// TwinCAT 3 PLC project Nepionic_PackML
// Title: Nepionic_PackML
// Company: Nepionic
// Author: Nepionic
// ProjectVersion: 0.1.1
// ProgramVersion: 3.1.4026.21
// libraries:
//   Nepionic_Log, * (Nepionic)
//   Tc2_System, * (Beckhoff Automation GmbH)
// project tree:
//   Commands/Generic/ ActionStateCommands.TcIO, HoldableStateCommands.TcIO, ClearedStateCommands.TcIO, ResettableStateCommands.TcIO, RunningStateCommands.TcIO
//   Commands/ AbortedCommands.TcIO, AbortingCommands.TcIO, ClearingCommands.TcIO, CompletedCommands.TcIO, CompletingCommands.TcIO, ExecuteCommands.TcIO, HeldCommands.TcIO, HoldingCommands.TcIO, IdleCommands.TcIO, ResettingCommands.TcIO, StartingCommands.TcIO, StoppedCommands.TcIO, StoppingCommands.TcIO, SuspendedCommands.TcIO, SuspendingCommands.TcIO, UnholdingCommands.TcIO, UnsuspendingCommands.TcIO
//   StateMachine/ State.TcDUT, StateMachine.TcPOU
//   UnitMode/ UnitMode.TcIO, DefaultUnitMode.TcPOU

// ---- StateMachine/State.TcDUT
{attribute 'qualified_only'}
{attribute 'strict'}
{attribute 'to_string'}
TYPE State :
(
	Undefined := 0,
    Clearing := 1,
    Stopped := 2,
    Starting := 3,
    Idle := 4,
    Suspended := 5,
	Execute := 6,
    Stopping := 7,
    Aborting := 8,
    Aborted := 9,
    Holding := 10,
    Held := 11,
    Unholding := 12,
    Suspending := 13,
    Unsuspending := 14,
    Resetting := 15,
    Completing := 16,
    Completed := 17
);
END_TYPE

// ---- Commands/Generic/ActionStateCommands.TcIO
INTERFACE PUBLIC ActionStateCommands EXTENDS __System.IQueryInterface

METHOD PUBLIC StateComplete
END_METHOD

END_INTERFACE

// ---- Commands/Generic/HoldableStateCommands.TcIO
INTERFACE PUBLIC HoldableStateCommands EXTENDS __System.IQueryInterface

METHOD PUBLIC Hold
END_METHOD

END_INTERFACE

// ---- Commands/Generic/ClearedStateCommands.TcIO
INTERFACE PUBLIC ClearedStateCommands EXTENDS __System.IQueryInterface

METHOD PUBLIC Abort
END_METHOD

END_INTERFACE

// ---- Commands/Generic/ResettableStateCommands.TcIO
INTERFACE PUBLIC ResettableStateCommands EXTENDS __System.IQueryInterface

METHOD PUBLIC Reset
END_METHOD

END_INTERFACE

// ---- Commands/Generic/RunningStateCommands.TcIO
INTERFACE PUBLIC RunningStateCommands EXTENDS ClearedStateCommands

METHOD PUBLIC Stop
END_METHOD

END_INTERFACE

// ---- Commands/AbortedCommands.TcIO
INTERFACE PUBLIC AbortedCommands EXTENDS __System.IQueryInterface

METHOD PUBLIC Clear
END_METHOD

END_INTERFACE

// ---- Commands/AbortingCommands.TcIO
INTERFACE PUBLIC AbortingCommands EXTENDS ActionStateCommands

END_INTERFACE

// ---- Commands/ClearingCommands.TcIO
INTERFACE PUBLIC ClearingCommands EXTENDS ClearedStateCommands, ActionStateCommands

END_INTERFACE

// ---- Commands/CompletedCommands.TcIO
INTERFACE PUBLIC CompletedCommands EXTENDS RunningStateCommands, ResettableStateCommands

END_INTERFACE

// ---- Commands/CompletingCommands.TcIO
INTERFACE PUBLIC CompletingCommands EXTENDS RunningStateCommands, ActionStateCommands

END_INTERFACE

// ---- Commands/ExecuteCommands.TcIO
INTERFACE PUBLIC ExecuteCommands EXTENDS RunningStateCommands, ActionStateCommands, HoldableStateCommands

METHOD PUBLIC Suspend
END_METHOD

END_INTERFACE

// ---- Commands/HeldCommands.TcIO
INTERFACE PUBLIC HeldCommands EXTENDS RunningStateCommands

METHOD PUBLIC Unhold
END_METHOD

END_INTERFACE

// ---- Commands/HoldingCommands.TcIO
INTERFACE PUBLIC HoldingCommands EXTENDS RunningStateCommands, ActionStateCommands

END_INTERFACE

// ---- Commands/IdleCommands.TcIO
INTERFACE PUBLIC IdleCommands EXTENDS RunningStateCommands

METHOD PUBLIC Start
END_METHOD

END_INTERFACE

// ---- Commands/ResettingCommands.TcIO
INTERFACE PUBLIC ResettingCommands EXTENDS RunningStateCommands, ActionStateCommands

END_INTERFACE

// ---- Commands/StartingCommands.TcIO
INTERFACE PUBLIC StartingCommands EXTENDS RunningStateCommands, ActionStateCommands, HoldableStateCommands

END_INTERFACE

// ---- Commands/StoppedCommands.TcIO
INTERFACE PUBLIC StoppedCommands EXTENDS ClearedStateCommands, ResettableStateCommands

END_INTERFACE

// ---- Commands/StoppingCommands.TcIO
INTERFACE PUBLIC StoppingCommands EXTENDS ClearedStateCommands, ActionStateCommands

END_INTERFACE

// ---- Commands/SuspendedCommands.TcIO
INTERFACE PUBLIC SuspendedCommands EXTENDS RunningStateCommands, HoldableStateCommands

METHOD PUBLIC Unsuspend
END_METHOD

END_INTERFACE

// ---- Commands/SuspendingCommands.TcIO
INTERFACE PUBLIC SuspendingCommands EXTENDS RunningStateCommands, ActionStateCommands, HoldableStateCommands

END_INTERFACE

// ---- Commands/UnholdingCommands.TcIO
INTERFACE PUBLIC UnholdingCommands EXTENDS RunningStateCommands, ActionStateCommands, HoldableStateCommands

END_INTERFACE

// ---- Commands/UnsuspendingCommands.TcIO
INTERFACE PUBLIC UnsuspendingCommands EXTENDS RunningStateCommands, ActionStateCommands, HoldableStateCommands

END_INTERFACE

// ---- UnitMode/UnitMode.TcIO
INTERFACE PUBLIC UnitMode

METHOD PUBLIC Abort
END_METHOD

METHOD PUBLIC Clear
END_METHOD

{attribute 'monitoring':='call'}
PROPERTY PUBLIC CurrentState : State
GET
END_GET
END_PROPERTY

METHOD PUBLIC CyclicCall
END_METHOD

METHOD PUBLIC Hold
END_METHOD

{attribute 'monitoring':='call'}
PROPERTY PUBLIC IsAborted : BOOL
GET
END_GET
END_PROPERTY

{attribute 'monitoring':='call'}
PROPERTY PUBLIC IsAborting : BOOL
GET
END_GET
END_PROPERTY

{attribute 'monitoring':='call'}
PROPERTY PUBLIC IsClearing : BOOL
GET
END_GET
END_PROPERTY

{attribute 'monitoring':='call'}
PROPERTY PUBLIC IsCompleted : BOOL
GET
END_GET
END_PROPERTY

{attribute 'monitoring':='call'}
PROPERTY PUBLIC IsCompleting : BOOL
GET
END_GET
END_PROPERTY

{attribute 'monitoring':='call'}
PROPERTY PUBLIC IsExecuting : BOOL
GET
END_GET
END_PROPERTY

{attribute 'monitoring':='call'}
PROPERTY PUBLIC IsHeld : BOOL
GET
END_GET
END_PROPERTY

{attribute 'monitoring':='call'}
PROPERTY PUBLIC IsHolding : BOOL
GET
END_GET
END_PROPERTY

{attribute 'monitoring':='call'}
PROPERTY PUBLIC IsIdle : BOOL
GET
END_GET
END_PROPERTY

{attribute 'monitoring':='call'}
PROPERTY PUBLIC IsResetting : BOOL
GET
END_GET
END_PROPERTY

{attribute 'monitoring':='call'}
PROPERTY PUBLIC IsStarting : BOOL
GET
END_GET
END_PROPERTY

{attribute 'monitoring':='call'}
PROPERTY PUBLIC IsStopped : BOOL
GET
END_GET
END_PROPERTY

{attribute 'monitoring':='call'}
PROPERTY PUBLIC IsStopping : BOOL
GET
END_GET
END_PROPERTY

{attribute 'monitoring':='call'}
PROPERTY PUBLIC IsSuspended : BOOL
GET
END_GET
END_PROPERTY

{attribute 'monitoring':='call'}
PROPERTY PUBLIC IsSuspending : BOOL
GET
END_GET
END_PROPERTY

{attribute 'monitoring':='call'}
PROPERTY PUBLIC IsUnholding : BOOL
GET
END_GET
END_PROPERTY

{attribute 'monitoring':='call'}
PROPERTY PUBLIC IsUnsuspending : BOOL
GET
END_GET
END_PROPERTY

METHOD PUBLIC Reset
END_METHOD

METHOD PUBLIC Start
END_METHOD

METHOD PUBLIC Stop
END_METHOD

METHOD PUBLIC Suspend
END_METHOD

METHOD PUBLIC Unhold
END_METHOD

METHOD PUBLIC Unsuspend
END_METHOD

END_INTERFACE

// ---- StateMachine/StateMachine.TcPOU
{attribute 'linkalways'} 
{attribute 'no_explicit_call' := 'This FB is a CLASS and must be accessed using methods or properties'}
{attribute 'enable_dynamic_creation'}
FUNCTION_BLOCK PUBLIC StateMachine
VAR_GENERIC CONSTANT
	initial_state : State := State.Idle;
END_VAR
IMPLEMENTS
	AbortingCommands,
	ClearingCommands,
	HeldCommands,
	CompletingCommands,
	ExecuteCommands,
	AbortedCommands,
	CompletedCommands,
	HoldingCommands,
	UnsuspendingCommands,
	UnholdingCommands,
	SuspendingCommands,
	SuspendedCommands,
	IdleCommands,
	ResettingCommands,
	StartingCommands,
	StoppedCommands,
	StoppingCommands
VAR
	current_state : State := initial_state;
	logger : DefaultLogger(__POUNAME());
END_VAR

METHOD PUBLIC Abort
IF IsAborting OR IsAborted THEN
	RETURN;
END_IF

logger.Debug('Abort() called, aborting');
ChangeState(State.Aborting);
END_METHOD

METHOD PRIVATE ChangeState
VAR_INPUT
	state : State;
END_VAR
logger
	.WithIntAttribute('exiting_state', current_state)
	.WithIntAttribute('entering_state', state)
	.Debug('Changing state');

current_state := state;
END_METHOD

METHOD PUBLIC Clear
IF IsAborted THEN
	logger.Debug('Clear() called, clearing');
	ChangeState(State.Clearing);
END_IF
END_METHOD

{attribute 'monitoring':='call'}
PROPERTY PUBLIC CurrentState : State
GET
CurrentState := current_state;
END_GET
END_PROPERTY

METHOD PUBLIC Hold
CASE current_state OF
	State.Execute,
	State.Starting,
	State.Suspending,
	State.Suspended,
	State.Unsuspending,
	State.Unholding:
		logger.Debug('Hold() called, holding');
		ChangeState(State.Holding);	
END_CASE
END_METHOD

{attribute 'monitoring':='call'}
PROPERTY PUBLIC IsAborted : BOOL
GET
IsAborted := (current_state = State.Aborted);
END_GET
END_PROPERTY

{attribute 'monitoring':='call'}
PROPERTY PUBLIC IsAborting : BOOL
GET
IsAborting := (current_state = State.Aborting);
END_GET
END_PROPERTY

{attribute 'monitoring':='call'}
PROPERTY PUBLIC IsClearing : BOOL
GET
IsClearing := (current_state = State.Clearing);
END_GET
END_PROPERTY

{attribute 'monitoring':='call'}
PROPERTY PUBLIC IsCompleted : BOOL
GET
IsCompleted := (current_state = State.Completed);
END_GET
END_PROPERTY

{attribute 'monitoring':='call'}
PROPERTY PUBLIC IsCompleting : BOOL
GET
IsCompleting := (current_state = State.Completing);
END_GET
END_PROPERTY

{attribute 'monitoring':='call'}
PROPERTY PUBLIC IsExecuting : BOOL
GET
IsExecuting := (current_state = State.Execute);
END_GET
END_PROPERTY

{attribute 'monitoring':='call'}
PROPERTY PUBLIC IsHeld : BOOL
GET
IsHeld := (current_state = State.Held);
END_GET
END_PROPERTY

{attribute 'monitoring':='call'}
PROPERTY PUBLIC IsHolding : BOOL
GET
IsHolding := (current_state = State.Holding);
END_GET
END_PROPERTY

{attribute 'monitoring':='call'}
PROPERTY PUBLIC IsIdle : BOOL
GET
isIdle := (current_state = State.Idle);
END_GET
END_PROPERTY

{attribute 'monitoring':='call'}
PROPERTY PUBLIC IsResetting : BOOL
GET
IsResetting := (current_state = State.Resetting);
END_GET
END_PROPERTY

{attribute 'monitoring':='call'}
PROPERTY PUBLIC IsStarting : BOOL
GET
IsStarting := (current_state = State.Starting);
END_GET
END_PROPERTY

{attribute 'monitoring':='call'}
PROPERTY PUBLIC IsStopped : BOOL
GET
isStopped := (current_state = State.Stopped);
END_GET
END_PROPERTY

{attribute 'monitoring':='call'}
PROPERTY PUBLIC IsStopping : BOOL
GET
IsStopping := (current_state = State.Stopping);
END_GET
END_PROPERTY

{attribute 'monitoring':='call'}
PROPERTY PUBLIC IsSuspended : BOOL
GET
IsSuspended := (current_state = State.Suspended);
END_GET
END_PROPERTY

{attribute 'monitoring':='call'}
PROPERTY PUBLIC IsSuspending : BOOL
GET
IsSuspending := (current_state = State.Suspending);
END_GET
END_PROPERTY

{attribute 'monitoring':='call'}
PROPERTY PUBLIC IsUnholding : BOOL
GET
IsUnholding := (current_state = State.Unholding);
END_GET
END_PROPERTY

{attribute 'monitoring':='call'}
PROPERTY PUBLIC IsUnsuspending : BOOL
GET
IsUnsuspending := (current_state = State.Unsuspending);
END_GET
END_PROPERTY

METHOD PUBLIC Reset
IF IsStopped OR IsCompleted THEN
	logger.Debug('Reset() called, resetting');
	ChangeState(State.Resetting);
END_IF
END_METHOD

METHOD PUBLIC Start
IF IsIdle THEN
	logger.Debug('Start() called, starting');
	ChangeState(State.Starting);
END_IF
END_METHOD

METHOD PUBLIC StateComplete
CASE current_state OF
	State.Idle: RETURN;
	State.Completed: RETURN;
	State.Stopped: RETURN;
	State.Held: RETURN;
	State.Suspended: RETURN;
	State.Aborted: RETURN;
END_CASE

logger.Debug('StateComplete() called, changing to new state');

CASE current_state OF
	State.Starting: ChangeState(State.Execute);
	State.Execute: ChangeState(State.Completing);
	State.Completing: ChangeState(State.Completed);
	State.Stopping: ChangeState(State.Stopped);
	State.Resetting: ChangeState(State.Idle);
	State.Holding: ChangeState(State.Held);
	State.Unholding: ChangeState(State.Execute);
	State.Suspending: ChangeState(State.Suspended);
	State.Unsuspending: ChangeState(State.Execute);
	State.Clearing: ChangeState(State.Stopped);
	State.Aborting: ChangeState(State.Aborted);
END_CASE
END_METHOD

METHOD PUBLIC Stop
CASE current_state OF
	State.Stopped: RETURN;
	State.Stopping: RETURN;
	State.Clearing: RETURN;
	State.Aborted: RETURN;
	State.Aborting: RETURN;
END_CASE

logger.Debug('Stop() called, stopping');
ChangeState(State.Stopping);
END_METHOD

METHOD PUBLIC Suspend
IF IsExecuting THEN 
	logger.Debug('Suspend() called, suspending');
	ChangeState(State.Suspending);
END_IF
END_METHOD

METHOD PUBLIC Unhold
IF IsHeld THEN
	logger.Debug('Unhold() called, unholding');
	ChangeState(State.Unholding);
END_IF
END_METHOD

METHOD PUBLIC Unsuspend
IF IsSuspended THEN
	logger.Debug('Unsuspend() called, unsuspending');
	ChangeState(State.Unsuspending);
END_IF
END_METHOD

END_FUNCTION_BLOCK

// ---- UnitMode/DefaultUnitMode.TcPOU
{attribute 'linkalways'} 
{attribute 'no_explicit_call' := 'This FB is a CLASS and must be accessed using methods or properties'}
{attribute 'enable_dynamic_creation'}
FUNCTION_BLOCK PUBLIC ABSTRACT DefaultUnitMode
VAR_GENERIC CONSTANT
	initial_state : State := State.Idle;
END_VAR
IMPLEMENTS UnitMode
VAR
	state_machine : StateMachine<initial_state>;
END_VAR

METHOD PUBLIC Abort
state_machine.Abort();
END_METHOD

METHOD PROTECTED Aborted
VAR_INPUT
	commands : AbortedCommands;
END_VAR
END_METHOD

METHOD PROTECTED Aborting
VAR_INPUT
	commands : AbortingCommands;
END_VAR
commands.StateComplete();
END_METHOD

METHOD PUBLIC Clear
state_machine.Clear();
END_METHOD

METHOD PROTECTED Clearing
VAR_INPUT
	commands : ClearingCommands;
END_VAR
commands.StateComplete();
END_METHOD

METHOD PROTECTED Completed
VAR_INPUT
	commands : CompletedCommands;
END_VAR
END_METHOD

METHOD PROTECTED Completing
VAR_INPUT
	commands : CompletingCommands;
END_VAR
commands.StateComplete();
END_METHOD

{attribute 'monitoring':='call'}
PROPERTY PUBLIC CurrentState : State
GET
CurrentState := state_machine.CurrentState;
END_GET
END_PROPERTY

METHOD PUBLIC CyclicCall
IF state_machine.IsIdle THEN 
	Idle(state_machine);
END_IF

IF state_machine.IsStarting THEN
	Starting(state_machine);
END_IF

IF state_machine.IsExecuting THEN
	Execute(state_machine);
END_IF

IF state_machine.IsCompleting THEN
	Completing(state_machine);
END_IF

IF state_machine.IsCompleted THEN
	Completed(state_machine);
END_IF

IF state_machine.IsStopping THEN
	Stopping(state_machine);
END_IF

IF state_machine.IsStopped THEN
	Stopped(state_machine);
END_IF

IF state_machine.IsResetting THEN
	Resetting(state_machine);
END_IF

IF state_machine.IsHolding THEN
	Holding(state_machine);
END_IF

IF state_machine.IsHeld THEN
	Held(state_machine);
END_IF

IF state_machine.IsUnholding THEN
	Unholding(state_machine);
END_IF

IF state_machine.IsSuspending THEN
	Suspending(state_machine);
END_IF

IF state_machine.IsSuspended THEN
	Suspended(state_machine);
END_IF

IF state_machine.IsUnsuspending THEN
	Unsuspending(state_machine);
END_IF

IF state_machine.IsClearing THEN
	Clearing(state_machine);
END_IF

IF state_machine.IsAborted THEN
	Aborted(state_machine);
END_IF

IF state_machine.IsAborting THEN
	Aborting(state_machine);
END_IF
END_METHOD

METHOD PROTECTED Execute
VAR_INPUT
	commands : ExecuteCommands;
END_VAR
commands.StateComplete();
END_METHOD

METHOD PROTECTED Held
VAR_INPUT
	commands : HeldCommands;
END_VAR
END_METHOD

METHOD PUBLIC Hold
state_machine.Hold();
END_METHOD

METHOD PROTECTED Holding
VAR_INPUT
	commands : HoldingCommands;
END_VAR
commands.StateComplete();
END_METHOD

METHOD PROTECTED Idle
VAR_INPUT
	commands : IdleCommands;
END_VAR
END_METHOD

{attribute 'monitoring':='call'}
PROPERTY PUBLIC IsAborted : bool
GET
IsAborted := state_machine.IsAborted;
END_GET
END_PROPERTY

{attribute 'monitoring':='call'}
PROPERTY PUBLIC IsAborting : bool
GET
IsAborting := state_machine.IsAborting;
END_GET
END_PROPERTY

{attribute 'monitoring':='call'}
PROPERTY PUBLIC IsClearing : bool
GET
IsClearing := state_machine.IsClearing;
END_GET
END_PROPERTY

{attribute 'monitoring':='call'}
PROPERTY PUBLIC IsCompleted : bool
GET
IsCompleted := state_machine.IsCompleted;
END_GET
END_PROPERTY

{attribute 'monitoring':='call'}
PROPERTY PUBLIC IsCompleting : bool
GET
IsCompleting := state_machine.IsCompleting;
END_GET
END_PROPERTY

{attribute 'monitoring':='call'}
PROPERTY PUBLIC IsExecuting : bool
GET
IsExecuting := state_machine.IsExecuting;
END_GET
END_PROPERTY

{attribute 'monitoring':='call'}
PROPERTY PUBLIC IsHeld : bool
GET
IsHeld := state_machine.IsHeld;
END_GET
END_PROPERTY

{attribute 'monitoring':='call'}
PROPERTY PUBLIC IsHolding : bool
GET
IsHolding := state_machine.IsHolding;
END_GET
END_PROPERTY

{attribute 'monitoring':='call'}
PROPERTY PUBLIC IsIdle : BOOL
GET
isIdle := state_machine.isIdle;
END_GET
END_PROPERTY

{attribute 'monitoring':='call'}
PROPERTY PUBLIC IsResetting : bool
GET
IsResetting := state_machine.IsResetting;
END_GET
END_PROPERTY

{attribute 'monitoring':='call'}
PROPERTY PUBLIC IsStarting : bool
GET
IsStarting := state_machine.IsStarting;
END_GET
END_PROPERTY

{attribute 'monitoring':='call'}
PROPERTY PUBLIC IsStopped : BOOL
GET
isStopped := state_machine.isStopped;
END_GET
END_PROPERTY

{attribute 'monitoring':='call'}
PROPERTY PUBLIC IsStopping : bool
GET
IsStopping := state_machine.IsStopping;
END_GET
END_PROPERTY

{attribute 'monitoring':='call'}
PROPERTY PUBLIC IsSuspended : bool
GET
IsSuspended := state_machine.IsSuspended;
END_GET
END_PROPERTY

{attribute 'monitoring':='call'}
PROPERTY PUBLIC IsSuspending : bool
GET
IsSuspending := state_machine.IsSuspending;
END_GET
END_PROPERTY

{attribute 'monitoring':='call'}
PROPERTY PUBLIC IsUnholding : bool
GET
IsUnholding := state_machine.IsUnholding;
END_GET
END_PROPERTY

{attribute 'monitoring':='call'}
PROPERTY PUBLIC IsUnsuspending : bool
GET
IsUnsuspending := state_machine.IsUnsuspending;
END_GET
END_PROPERTY

METHOD PUBLIC Reset
state_machine.Reset();
END_METHOD

METHOD PROTECTED Resetting
VAR_INPUT
	commands : ResettingCommands;
END_VAR
commands.StateComplete();
END_METHOD

METHOD PUBLIC Start
state_machine.Start();
END_METHOD

METHOD PROTECTED Starting
VAR_INPUT
	commands : StartingCommands;
END_VAR
commands.StateComplete();
END_METHOD

METHOD PUBLIC Stop
state_machine.Stop();
END_METHOD

METHOD PROTECTED Stopped
VAR_INPUT
	commands : StoppedCommands;
END_VAR
END_METHOD

METHOD PROTECTED Stopping
VAR_INPUT
	commands : StoppingCommands;
END_VAR
commands.StateComplete();
END_METHOD

METHOD PUBLIC Suspend
state_machine.Suspend();
END_METHOD

METHOD PROTECTED Suspended
VAR_INPUT
	commands : SuspendedCommands;
END_VAR
END_METHOD

METHOD PROTECTED Suspending
VAR_INPUT
	commands : SuspendingCommands;
END_VAR
commands.StateComplete();
END_METHOD

METHOD PUBLIC Unhold
state_machine.Unhold();
END_METHOD

METHOD PROTECTED Unholding
VAR_INPUT
	commands : UnholdingCommands;
END_VAR
commands.StateComplete();
END_METHOD

METHOD PUBLIC Unsuspend
state_machine.Unsuspend();
END_METHOD

METHOD PROTECTED Unsuspending
VAR_INPUT
	commands : UnsuspendingCommands;
END_VAR
commands.StateComplete();
END_METHOD

END_FUNCTION_BLOCK
